{attribute 'qualified_only'}
{attribute 'strict'}
TYPE System_Modus_Enum :
(
	System_Init := 0,
	System_Run
);
END_TYPE

(* stored: Version 1.1.0.1, ProductVersion 3.1.4024.13
   DUT System_Modus_Enum: Id {7dae0757-e2ec-40c7-a7b0-86cf54e4e073} *)
